Fanuc KAREL source: kt00010.KL

-- PROVISIONAL review KL for V770-1; original PC SHA256 eb57a37db6a6f42bc93fa3a7f7a3142c8cd41e6d619affc5a018c7f3ab8213da
-- Incomplete behavior may be omitted. Consult companion uncertainty JSON. Do not deploy.
PROGRAM KT00010
%NOLOCKGROUP
VAR
  R1 : REAL
  I2 : INTEGER
  OUT : REAL
BEGIN
  -- UNRESOLVED_PC offsets 5-16; opcodes 2E,23
  -- UNRESOLVED_PC offsets 21-32; opcodes 2E,23
  -- UNRESOLVED_PC offsets 37-57; opcodes 21,21,64,69,23
  -- UNRESOLVED_PC offsets 62-66; opcodes 7F
END KT00010
